// TIA Portal V17 export
// export: Created 2025-03-07T09:24:36.7959296Z, ExportSetting WithDefaults, DisplayName Totally Integrated Automation Portal, DisplayVersion V17 Update 8, DisplayName TIA Portal Openness, DisplayVersion V17 Update 8, DisplayName TIA Portal Version Control Interface, DisplayVersion V17, DisplayName SINAMICS Startdrive Advanced, DisplayVersion V17 SP2, DisplayName SINAMICS Startdrive G110M, G120, G120C, G120D, G120P, G115D, DisplayVersion V17 SP2, DisplayName SINAMICS Startdrive G130, G150, S120, S150, SINAMICS MV, S210, DisplayVersion V17 SP2, DisplayName STEP 7 Professional, DisplayVersion V17 Update 8, DisplayName SINUMERIK ONE STEP 7 Toolbox, DisplayVersion V17 Update 12, DisplayName SINUMERIK 840D sl STEP 7 Toolbox, DisplayVersion V17 Update 12, DisplayName STEP 7 Safety, DisplayVersion V17 Update 6, DisplayName WinCC Advanced, DisplayVersion V17 Update 8
TYPE "GENERAL_DATA_START_STOP"
// stored: IsFailsafeCompliant false
   STRUCT
      START_GENERAL_CONDITIONS : Bool;   // Start general conditions
      START_GENERAL_CONDITIONS_HELP : Bool;   // Start general conditions help
      START_INITIAL_CONDITIONS : Bool;   // Start initial conditions
      START_INITIAL_CONDITIONS_HELP : Bool;   // Start initial conditions help
      START_MANUAL_REQUEST : Bool;   // Start manual request
      START_SEMI_REQUEST : Bool;   // Start semi request
      START_AUTO_REQUEST : Bool;   // Start auto request
      START_GLOBAL_REQUEST : Bool;   // Start global request
      START_COMMAND : Bool;   // Start command
      FEEDBACK_ON : Bool;   // Feedback on
      SYSTEM_ON : Bool;   // System on
      STOP_GENERAL_CONDITIONS : Bool;   // Stop general conditions
      STOP_GENERAL_CONDITIONS_HELP : Bool;   // Stop general conditions help
      STOP_INITIAL_CONDITIONS : Bool;   // Stop initial conditions
      STOP_INITIAL_CONDITIONS_HELP : Bool;   // Stop initial conditions help
      STOP_MANUAL_REQUEST : Bool;   // Stop manual request
      STOP_SEMI_REQUEST : Bool;   // Stop semi request
      STOP_AUTO_REQUEST : Bool;   // Stop auto request
      STOP_GLOBAL_REQUEST : Bool;   // Stop global request
      STOP_COMMAND : Bool;   // Stop command
      FEEDBACK_OFF : Bool;   // Feedback off
      SYSTEM_OFF : Bool;   // System off
      FAULT : Bool;   // Fault
   END_STRUCT;
END_TYPE
